{attribute 'pack_mode' := '1'}
TYPE
  ST_OpcUa_UintPointWrite :
  STRUCT
    ErrorCode : UDINT;
    Value : UINT;
  END_STRUCT
END_TYPE

(* stored: Version 1.1.0.1, ProductVersion 3.1.4024.9
   DUT ST_OpcUa_UintPointWrite: Id {6d8bd1f7-2406-43b6-9ba3-ad4d62a74481} *)
